// TwinCAT 3 PLC project RobotArmPLC
// ProgramVersion: 3.1.0.8
// libraries:
//   Tc2_MC2, * (Beckhoff Automation GmbH)
//   Tc2_SerialCom, * (Beckhoff Automation GmbH)
//   Tc2_Standard, * (Beckhoff Automation GmbH)
//   Tc2_System, * (Beckhoff Automation GmbH)
//   Tc3_Interfaces, * (Beckhoff Automation GmbH)
//   Tc3_Module, * (Beckhoff Automation GmbH)
// project tree:
//   GVLs/ GVL.TcGVL
//   / PlcTask.TcTTO
//   POUs/ MAIN.TcPOU, SerialRecieve.TcPOU, ShoudlerInit.TcPOU, ShoulderLevelShift.TcPOU, ShoulderRotate.TcPOU
// real-time tasks:
//   TASK PlcTask: cycle T#10ms, priority 20, ADS port 350
//   TASK CPP: cycle T#10ms, priority 1, ADS port 351
// motion (NC):
//   TASK NC-Task 1 SAF: cycle T#10ms, priority 4, ADS port 501
//   TASK NC-Task 1 SVB: cycle T#10ms, priority 8, ADS port 511
//   AXIS AxisShoulderLevelShift (id 1)
//     Velo: SlowManual=0.5, FastManual=2, Maximum=8
//     OtherSettings: AllowMotionCmdToSlave=true
//     encoder EncType=19
//       EncPara: MaxCount=#xffffffff
//     drive DrvType=16
//       DrvPara: MaxCount=#xffffffff
//         Analog: VeloReferenz=7
//         TimeComp: TaskDelayCycles=1
//     controller CtrType=1
//       CtrPara: PriorControlFactor=1
//         Observer: BandWidth=20
//   AXIS AxisShoulderRotate (id 2)
//     Velo: SlowManual=0.5, FastManual=2, Maximum=8
//     OtherSettings: AllowMotionCmdToSlave=true
//     encoder EncType=19
//       EncPara: MaxCount=#xffffffff
//     drive DrvType=16
//       DrvPara: MaxCount=#xffffffff
//         Analog: VeloReferenz=7
//         TimeComp: TaskDelayCycles=1
//     controller CtrType=1
//       CtrPara: PriorControlFactor=1
//         Observer: BandWidth=20
// I/O:
//   DEVICE Device 1 (EtherCAT), AmsNetId 5.36.3.8.2.1
//     Term 1 (EK1200) [EK1200-5000 EtherCAT Power supply (2A E-Bus)]
//       Term 2 (EL2502) [EL2502 2Ch. PWM output, 24V]
//       Term 3 (EL6001) [EL6001 Interface (RS232)]
//       Term 4 (EL4102) [EL4102 2Ch. Ana. Output  0-10V, 16bit]
//       Term 5 (EL2502) [EL2502 2K. PWM Ausgang, 24V]
//       Term 6 (EL2502) [EL2502 2Ch. PWM Output, 24V]
//       Term 7 (EL2502) [EL2502 2Ch. PWM Output, 24V]
//       Term 8 (EL3008) [EL3008 8Ch. Ana. Input +/-10V]
//       Term 9 (EL2502) [EL2502 2Ch. PWM output, 24V]
//       Term 10 (EL2502) [EL2502 2K. PWM Ausgang, 24V]
//       Term 11 (EL2502) [EL2502 2K. PWM Ausgang, 24V]
//       Term 12 (EL2502) [EL2502 2Ch. PWM output, 24V]
//       Term 13 (EL3692) [EL3692 2Ch. resistance measurement terminal]
//       Term 14 (EL9011) [EL9011 End Terminal]
//   DEVICE Device 4 (EtherCAT), AmsNetId 5.36.3.8.5.1
//     Drive 1 (Elmo Drive) [Gold EtherCAT GCON Drive Rev:0x000103F6]
//     Drive 2 (Elmo Drive) [Gold EtherCAT GCON Drive Rev:0x000103F6]
// variable links:
//   Device 1 (EtherCAT) <-> RobotArmCPP/RobotArmCPP_Obj1 (CRobotArmMain)
//     Term 1 (EK1200)/Term 10 (EL2502)/PWM Outputs Channel 1/PWM output <-> Outputs/wrist_three
//     Term 1 (EK1200)/Term 10 (EL2502)/PWM Outputs Channel 2/PWM output <-> Outputs/wrist_four
//     Term 1 (EK1200)/Term 11 (EL2502)/PWM Outputs Channel 1/PWM output <-> Outputs/wrist_five
//     Term 1 (EK1200)/Term 11 (EL2502)/PWM Outputs Channel 2/PWM output <-> Outputs/wrist_six
//     Term 1 (EK1200)/Term 12 (EL2502)/PWM Outputs Channel 1/PWM output <-> Outputs/wrist_seven
//     Term 1 (EK1200)/Term 12 (EL2502)/PWM Outputs Channel 2/PWM output <-> Outputs/wrist_eight
//     Term 1 (EK1200)/Term 13 (EL3692)/SAI Inputs Real Channel 1/Value <-> Inputs/wrist_resistor
//     Term 1 (EK1200)/Term 4 (EL4102)/Channel 1/Output <-> Outputs/ElbowOutM1
//     Term 1 (EK1200)/Term 4 (EL4102)/Channel 2/Output <-> Outputs/ElbowOutM2
//     Term 1 (EK1200)/Term 5 (EL2502)/PWM Outputs Channel 1/PWM output <-> Outputs/hand_one
//     Term 1 (EK1200)/Term 5 (EL2502)/PWM Outputs Channel 2/PWM output <-> Outputs/hand_two
//     Term 1 (EK1200)/Term 6 (EL2502)/PWM Outputs Channel 1/PWM output <-> Outputs/hand_three
//     Term 1 (EK1200)/Term 6 (EL2502)/PWM Outputs Channel 2/PWM output <-> Outputs/hand_four
//     Term 1 (EK1200)/Term 7 (EL2502)/PWM Outputs Channel 1/PWM output <-> Outputs/hand_fan
//     Term 1 (EK1200)/Term 8 (EL3008)/AI Standard Channel 1/Value <-> Inputs/hand_one_temp
//     Term 1 (EK1200)/Term 8 (EL3008)/AI Standard Channel 2/Value <-> Inputs/hand_two_temp
//     Term 1 (EK1200)/Term 8 (EL3008)/AI Standard Channel 3/Value <-> Inputs/hand_three_temp
//     Term 1 (EK1200)/Term 8 (EL3008)/AI Standard Channel 4/Value <-> Inputs/hand_four_temp
//     Term 1 (EK1200)/Term 9 (EL2502)/PWM Outputs Channel 1/PWM output <-> Outputs/wrist_one
//     Term 1 (EK1200)/Term 9 (EL2502)/PWM Outputs Channel 2/PWM output <-> Outputs/wrist_two
//   NC-Task 1 SAF/Axes/AxisShoulderLevelShift <-> Device 4 (EtherCAT)/Drive 1 (Elmo Drive)
//     Drive/Inputs/In/nDcOutputTime <-> InfoData/DcOutputShift
//     Drive/Inputs/In/nState1 <-> Inputs/Status word
//     Drive/Inputs/In/nState2 <-> Inputs/Status word @bit 8
//     Drive/Inputs/In/nState4 @bit 1 <-> WcState/InputToggle
//     Drive/Inputs/In/nState4 <-> WcState/WcState
//     Drive/Outputs/Out/nCtrl1 <-> Outputs/Control word
//     Drive/Outputs/Out/nCtrl2 <-> Outputs/Control word @bit 8
//     Drive/Outputs/Out/nDataOut1 <-> Outputs/Target Position
//     Enc/Inputs/In/nDataIn1 <-> Inputs/Position actual value
//     Enc/Inputs/In/nDcInputTime <-> InfoData/DcInputShift
//     Enc/Inputs/In/nState4 @bit 1 <-> WcState/InputToggle
//     Enc/Inputs/In/nState4 <-> WcState/WcState
//   NC-Task 1 SAF/Axes/AxisShoulderRotate <-> Device 4 (EtherCAT)/Drive 2 (Elmo Drive)
//     Drive/Inputs/In/nDcOutputTime <-> InfoData/DcOutputShift
//     Drive/Inputs/In/nState1 <-> Inputs/Status word
//     Drive/Inputs/In/nState2 <-> Inputs/Status word @bit 8
//     Drive/Inputs/In/nState4 @bit 1 <-> WcState/InputToggle
//     Drive/Inputs/In/nState4 <-> WcState/WcState
//     Drive/Outputs/Out/nCtrl1 <-> Outputs/Control word
//     Drive/Outputs/Out/nCtrl2 <-> Outputs/Control word @bit 8
//     Drive/Outputs/Out/nDataOut1 <-> Outputs/Target Position
//     Enc/Inputs/In/nDataIn1 <-> Inputs/Position actual value
//     Enc/Inputs/In/nDcInputTime <-> InfoData/DcInputShift
//     Enc/Inputs/In/nState4 @bit 1 <-> WcState/InputToggle
//     Enc/Inputs/In/nState4 <-> WcState/WcState
//   RobotArmPLC/RobotArmPLC Instance <-> Device 1 (EtherCAT)/Term 1 (EK1200)/Term 3 (EL6001)
//     PlcTask Inputs/SerialRecieve.EL6_22Bin_PC1/D <-> COM Inputs/Data In 0
//     PlcTask Inputs/SerialRecieve.EL6_22Bin_PC1/D @bit {8..168 step 8} <-> COM Inputs/Data In {1..21}  (21 links)
//     PlcTask Inputs/SerialRecieve.EL6_22Bin_PC1/Status <-> COM Inputs/Status
//     PlcTask Outputs/SerialRecieve.EL6_22Bout_PC1/Ctrl <-> COM Outputs/Ctrl
//     PlcTask Outputs/SerialRecieve.EL6_22Bout_PC1/D <-> COM Outputs/Data Out 0
//     PlcTask Outputs/SerialRecieve.EL6_22Bout_PC1/D @bit {8..168 step 8} <-> COM Outputs/Data Out {1..21}  (21 links)
//   RobotArmPLC/RobotArmPLC Instance <-> NC-Task 1 SAF/Axes/AxisShoulderLevelShift
//     PlcTask Inputs/GVL.AxisLevelShift.NcToPlc <-> Outputs/ToPlc
//     PlcTask Outputs/GVL.AxisLevelShift.PlcToNc <-> Inputs/FromPlc
//   RobotArmPLC/RobotArmPLC Instance <-> NC-Task 1 SAF/Axes/AxisShoulderRotate
//     PlcTask Inputs/GVL.AxisRotate.NcToPlc <-> Outputs/ToPlc
//     PlcTask Outputs/GVL.AxisRotate.PlcToNc <-> Inputs/FromPlc
//   RobotArmPLC/RobotArmPLC Instance <-> RobotArmCPP/RobotArmCPP_Obj1 (CRobotArmMain)
//     PlcTask Inputs/GVL.CppErrorCode <-> CppToPlc/ErrorCode
//     PlcTask Inputs/GVL.ShoulderInitStart <-> CppToPlc/ShoulderInitStart
//     PlcTask Inputs/MAIN.ElbowAngle <-> CppToPlc/ElbowAngle
//     PlcTask Inputs/MAIN.ElbowTarAngle <-> CppToPlc/ElbowTarAngle
//     PlcTask Inputs/MAIN.hand_four_pwm <-> CppToPlc/hand_four_pwm
//     PlcTask Inputs/MAIN.hand_four_temp <-> CppToPlc/hand_four_temp
//     PlcTask Inputs/MAIN.hand_one_temp <-> CppToPlc/hand_one_temp
//     PlcTask Inputs/MAIN.hand_onepwm <-> CppToPlc/hand_one_pwm
//     PlcTask Inputs/MAIN.hand_three_pwm <-> CppToPlc/hand_three_pwm
//     PlcTask Inputs/MAIN.hand_three_temp <-> CppToPlc/hand_three_temp
//     PlcTask Inputs/MAIN.hand_two_pwm <-> CppToPlc/hand_two_pwm
//     PlcTask Inputs/MAIN.hand_two_temp <-> CppToPlc/hand_two_temp
//     PlcTask Inputs/MAIN.wrist_angle <-> CppToPlc/wrist_angle
//     PlcTask Inputs/MAIN.wrist_error <-> CppToPlc/wrist_error
//     PlcTask Inputs/MAIN.wrist_pwm_out <-> CppToPlc/wrist_pwm
//     PlcTask Inputs/MAIN.wrist_tarAngle <-> CppToPlc/wrist_tarAngle
//     PlcTask Inputs/ShoulderLevelShift.TarPosLevelShift <-> CppToPlc/TarPosLevelShift
//     PlcTask Inputs/ShoulderRotate.TarPosRotate <-> CppToPlc/TarPosRotate
//     PlcTask Outputs/GVL.ChooseAction <-> PlcToCpp/ChooseAction
//     PlcTask Outputs/GVL.ExtEnabledLevelShift <-> PlcToCpp/LevelShiftExtEnabled
//     PlcTask Outputs/GVL.ExtEnabledRotate <-> PlcToCpp/RotateExtEnabled
//     PlcTask Outputs/GVL.IsRepeat <-> PlcToCpp/IsRepeat
//     PlcTask Outputs/GVL.PosLevelShift <-> PlcToCpp/PosLevelShift
//     PlcTask Outputs/GVL.PosRotate <-> PlcToCpp/PosRotate
//     PlcTask Outputs/GVL.SetTarAngle <-> PlcToCpp/SetTarAngle
//     PlcTask Outputs/GVL.SetTarSpeed <-> PlcToCpp/SetTarSpeed
//     PlcTask Outputs/GVL.ShoulderInitFinish <-> PlcToCpp/ShoulderInitFinish
//     PlcTask Outputs/GVL.StopElbow <-> PlcToCpp/StopElbow
//     PlcTask Outputs/GVL.StopHand <-> PlcToCpp/StopHand
//     PlcTask Outputs/GVL.StopWrist <-> PlcToCpp/StopWrist
//     PlcTask Outputs/GVL.Timer <-> PlcToCpp/Timer
//     PlcTask Outputs/MAIN.PlcStarted <-> PlcToCpp/PlcStarted
//     PlcTask Outputs/SerialRecieve.JIAODU <-> PlcToCpp/ElbowAngle

CONFIGURATION RobotArmPLC
    RESOURCE PLC ON TwinCAT3
        TASK PlcTask(INTERVAL := T#10ms, PRIORITY := 20);
        PROGRAM MAIN WITH PlcTask : MAIN;
        PROGRAM SerialRecieve WITH PlcTask : SerialRecieve;
        PROGRAM ShoudlerInit WITH PlcTask : ShoudlerInit;
        PROGRAM ShoulderLevelShift WITH PlcTask : ShoulderLevelShift;
        PROGRAM ShoulderRotate WITH PlcTask : ShoulderRotate;
    END_RESOURCE
END_CONFIGURATION

// ---- GVLs/GVL.TcGVL
VAR_GLOBAL
	//肩关节水平移动自由度变量
	AxisLevelShift: AXIS_REF;											//运动轴
	MC_PowerLevelShift: MC_Power;										//电源模块
	MC_MoveAbsoluteLevelShift: MC_MoveAbsolute;							//绝对运动模块
	PosLevelShift AT%Q* : LREAL;										//平移运动位置.输出给C++
	
	//肩关节旋转移动自由度变量
	AxisRotate: AXIS_REF;												//运动轴
	MC_PowerRotate: MC_Power;											//电源模块
	MC_MoveAbsoluteRotate: MC_MoveAbsolute;								//绝对运动模块
	MC_ExtSetPointGenDisableRotate: MC_ExtSetPointGenDisable;			//外部给定运动禁止
	MC_ExtSetPointGenEnableRotate: MC_ExtSetPointGenEnable;				//外部给定运动使能
	PosRotate AT%Q* : LREAL;											//旋转移动位置.输出给C++
	
	//肩关节初始化完成标志量
	ShoulderInitStart AT%I* : BOOL := FALSE;							//肩关节初始化启动
	ShoulderInitFinish AT%Q*: BOOL := FALSE;
	ExtEnabledLevelShift AT%Q* : BOOL := FALSE;							//平移外部给定模块已使能
	ExtEnabledRotate AT%Q* : BOOL := FALSE;								//旋转外部给定模块已使能
	
	//PLC时间
	Timer AT%Q*: LREAL := 0;											//时间 
	
	//错误记录
	CppErrorCode AT%I*: INT := 0;										//C++错误代码，在PLC显示，容易看到。
	ErrorCode: INT := 0;												//PLC错误代码，TODO:研究可持续写入的变量，类似字符串。
	ErrorTime: LREAL := 0;												//错误发生的时间，共4位
																		//第一位无意义，第二位表示关节（0-4：肩平移、肩旋转、肘、腕、手）
																		//第三位表示关节自由度（例如肩关节0表示平移自由度，1表示旋转自由度）
																		//第四位表示错误信息
																		//1000：平移初始化电源使能错误
																		//1001：平移位置超过限制
																		//1002：平移速度超过限制
																		//1100：旋转初始化电源使能错误
																		//1101：旋转位置超过限制
																		//1102：旋转速度超过限制
	ErrorTarPosLevelShift : LREAL := 0;									//错误发生时平移期望位置
	ErrorTarPosRotate : LREAL := 0;										//错误发生时旋转期望位置
	
	StopElbow AT%Q* : BOOL := FALSE;									//气动放气标志量，手动在plc里设置
	StopWrist AT%Q* : BOOL := FALSE;
	StopHand AT%Q* : BOOL := FALSE;
	
	ChooseAction AT%Q* : INT := -1;
	IsRepeat AT%Q* : BOOL := FALSE;
	SetTarAngle AT%Q* : LREAL := 30;									//角度定位
	SetTarSpeed AT%Q* : LREAL := 2;										//速度设置，到达100度
END_VAR

// ---- POUs/MAIN.TcPOU
PROGRAM MAIN
VAR
	ElbowTarAngle AT%I* : LREAL;
	ElbowAngle AT%I* : LREAL;
	ElbowAngleError : LREAL;
	PlcStarted AT%Q* : BOOL := FALSE;
	
	wrist_pwm_out AT%I*: LREAL;
	wrist_angle AT%I*: LREAL;
	wrist_tarAngle AT%I*: LREAL;
	wrist_error AT%I*: LREAL;
	flag_plc AT%Q*: BOOL;
///////////////腕关节变量监测/////
	
	hand_one_temp AT%I*: INT;
	hand_two_temp AT%I*: INT;
	hand_three_temp AT%I*: INT;
	hand_four_temp AT%I*: INT;
	hand_onepwm AT%I*: INT;
	hand_two_pwm AT%I*: INT;
	hand_three_pwm AT%I*: INT;
	hand_four_pwm AT%I*: INT;
/////////////手部变量监测/////////
END_VAR

//PlcStarted := TRUE;

(*IF InitFinish AND ExtEnabledLevelShift AND ExtEnabledRotate THEN
	Timer := Timer + 0.01;
END_IF*)
Timer := Timer + 0.01;

ElbowAngleError := ElbowTarAngle - ElbowAngle;
wrist_error := wrist_tarAngle - wrist_angle;

END_PROGRAM

// ---- POUs/SerialRecieve.TcPOU
PROGRAM SerialRecieve
VAR
	//读取编码器角度
	EL6_22Bin_PC1	AT %I* 	: KL6inData22b;
	EL6_22Bout_PC1	AT %Q*	: KL6outData22b;
	RxBuffer1: COMBuffer;
	TxBuffer1: COMBuffer;
	JIAODU	AT %Q* : LREAL;(*单位 度*)
	JIAOSUDU: LREAL;(*单位 度*)
	JIAOJIASUDU: LREAL;(*单位 度*)
	SerialLineControlElbow:SerialLineControl;
	
	i:INT;
    AA:BYTE;
	BB:BYTE;
	RxBufferStep:INT:=0;
    AA_P:BYTE;
	BB_P:BYTE;
	JIAODU_INT:INT;
	J1: LREAL:=0;
	J2: LREAL:=0;
	J3: LREAL:=0;
	W1: LREAL:=0;
	W2: LREAL:=0;
	t_tip: LREAL:=0.01;
END_VAR

//读取编码器的数值
SerialLineControlElbow(
	Mode:= SERIALLINEMODE_KL6_22B_STANDARD, 
	pComIn:= ADR(EL6_22Bin_PC1), 
	pComOut:= ADR(EL6_22Bout_PC1), 
	SizeComIn:= UINT_TO_INT(SIZEOF(EL6_22Bin_PC1)), 
	TxBuffer:= TxBuffer1, 
	RxBuffer:= RxBuffer1);

IF RxBuffer1.Count<> 0 THEN
	FOR i:=1 TO UINT_TO_INT(RxBuffer1.Count) DO
		IF RxBufferStep=3 THEN
			BB:=RxBuffer1.Buffer[RxBuffer1.RdIdx];
			AA:=AA_P;
			RxBufferStep:=0;
		END_IF
		IF RxBufferStep=2 THEN
			AA_P:=RxBuffer1.Buffer[RxBuffer1.RdIdx];
			RxBufferStep:=3;
		END_IF
		IF RxBufferStep=1 THEN
			IF RxBuffer1.Buffer[RxBuffer1.RdIdx]=90 THEN
				RxBufferStep:=2;
			ELSE
				RxBufferStep:=0;
			END_IF
		END_IF
		IF RxBuffer1.Buffer[RxBuffer1.RdIdx]=165 THEN
			RxBufferStep:=1;
		END_IF

		RxBuffer1.RdIdx:=RxBuffer1.RdIdx+1;
		IF RxBuffer1.RdIdx>300 THEN
			RxBuffer1.RdIdx:=0;
		END_IF
	END_FOR
RxBuffer1.Count:=0;
END_IF

JIAODU_INT:=UINT_TO_INT(AA*256+BB);
JIAODU:=INT_TO_REAL(JIAODU_INT)*360.0/4096.0;
J3:=J2;
J2:=J1;
J1:=JIAODU;
JIAOSUDU:=(J1-J2)/t_tip;
W2:=W1;
W1:=JIAOSUDU;
JIAOJIASUDU:=(W1-W2)/t_tip;

END_PROGRAM

// ---- POUs/ShoudlerInit.TcPOU
PROGRAM ShoudlerInit
VAR
	InitPosLevelShift: LREAL := 0;			//平移自由度.初始化位置
	InitStatusLevelShift: INT := 0;			//平移自由度.初始化状态变量	
	InitFinishLevelShift: BOOL := FALSE;	//平移自由度.初始化完成标志量
	
	InitPosRotate: LREAL := 0;				//旋转自由度.初始化位置
	InitStatusRotate: INT := 0;				//旋转自由度.初始化状态变量	
	InitFinishRotate: BOOL := FALSE;		//旋转自由度.初始化完成标志量
END_VAR

//肩关节初始化

//平移自由度
MC_PowerLevelShift(
	Axis:= AxisLevelShift,
	Enable_Positive:= TRUE,
	Enable_Negative:= TRUE, );
	
MC_MoveAbsoluteLevelShift(
	Axis:= AxisLevelShift, );

CASE InitStatusLevelShift OF
	0://等待初始化命令
		IF ShoulderInitStart THEN
			InitStatusLevelShift := 1;
		END_IF
	1://init 初始化
		MC_PowerLevelShift.Enable := FALSE;
		MC_MoveAbsoluteLevelShift.Execute := FALSE;
		InitStatusLevelShift := 2;
	2://power 使能
		MC_PowerLevelShift.Enable := TRUE;
		IF MC_PowerLevelShift.Status THEN
			InitStatusLevelShift := 3;
		END_IF
		IF AxisLevelShift.Status.Error THEN
			ErrorTime := Timer;
			InitStatusLevelShift := 5;
		END_IF
	3://move 移动到初始位置
		MC_MoveAbsoluteLevelShift.Position := InitPosLevelShift;
		MC_MoveAbsoluteLevelShift.Velocity := 1;
		MC_MoveAbsoluteLevelShift.Execute := TRUE;
		IF MC_MoveAbsoluteLevelShift.Done THEN
			MC_MoveAbsoluteLevelShift.Execute := FALSE;
			InitStatusLevelShift := 4;
		END_IF
	4://finishInit 初始化完成
		InitFinishLevelShift := TRUE;
	5://error
		ErrorCode := 1000;
END_CASE


//旋转自由度
MC_PowerRotate(
	Axis:= AxisRotate,
	Enable_Positive:= TRUE,
	Enable_Negative:= TRUE, );
	
MC_MoveAbsoluteRotate(
	Axis:= AxisRotate, );

CASE InitStatusRotate OF
	0://等待初始化命令
		IF ShoulderInitStart THEN
			InitStatusRotate := 1;
		END_IF
	1://init 初始化
		MC_PowerRotate.Enable := FALSE;
		MC_MoveAbsoluteRotate.Execute := FALSE;
		InitStatusRotate := 2;
	2://power 使能
		MC_PowerRotate.Enable := TRUE;
		IF MC_PowerRotate.Status THEN
			InitStatusRotate := 3;
		END_IF
		IF AxisLevelShift.Status.Error THEN
			ErrorTime := Timer;
			InitStatusRotate := 5;
		END_IF
	3://move 移动到初始位置
		MC_MoveAbsoluteRotate.Position := InitPosLevelShift;
		MC_MoveAbsoluteRotate.Velocity := 1;
		MC_MoveAbsoluteRotate.Execute := TRUE;
		IF MC_MoveAbsoluteRotate.Done THEN
			MC_MoveAbsoluteRotate.Execute := FALSE;
			InitStatusRotate := 4;
		END_IF
	4://finishInit 初始化完成
		InitFinishRotate := TRUE;
	5://error
		ErrorCode := 1100;
END_CASE
		
IF InitFinishLevelShift AND InitFinishRotate THEN
	ShoulderInitFinish := TRUE;
END_IF

END_PROGRAM

// ---- POUs/ShoulderLevelShift.TcPOU
PROGRAM ShoulderLevelShift
VAR
	MC_ExtSetPointGenDisableLevelShift: MC_ExtSetPointGenDisable;		//外部给定运动禁止
	MC_ExtSetPointGenEnableLevelShift: MC_ExtSetPointGenEnable;			//外部给定运动使能
	
	//TODO: C++将目标角度转换为目标位置
	TarPosLevelShift AT%I* : LREAL := 0;								//平移目标位置，C++给定
	ErrPosLevelShift: LREAL := 0;										//目标位置和实际位置误差
	
	StatusLevelShift: INT := 0;											//状态变量
	
	test : LREAL := 0;
END_VAR

//肩关节水平移动自由度

//电机外部给定运动模块参数设置
MC_ExtSetPointGenDisableLevelShift(
	Axis:= AxisLevelShift, );
	
MC_ExtSetPointGenEnableLevelShift(
	Axis:= AxisLevelShift, );
	
PosLevelShift := AxisLevelShift.NcToPlc.ActPos;

CASE StatusLevelShift OF
	0:	//判断是否完成初始化
		IF ShoulderInitFinish THEN
			StatusLevelShift := 1;
		END_IF
	1:	//外部给定模块使能给低电平
		MC_ExtSetPointGenEnableLevelShift.Execute := FALSE;
		MC_ExtSetPointGenDisableLevelShift.Execute := FALSE;
		StatusLevelShift := 2;
	2:
		MC_ExtSetPointGenEnableLevelShift.Execute := TRUE;
		IF MC_ExtSetPointGenEnableLevelShift.Enabled THEN
			StatusLevelShift := 3;
			ExtEnabledLevelShift := TRUE;
		END_IF
	3:	//判断目标移动是否有问题
		//Timer := Timer + 0.01;
		IF TarPosLevelShift > 18 OR TarPosLevelShift < -15 THEN
			ErrorCode := 1001;
			ErrorTime := Timer;
			StatusLevelShift := 4;						//跳转到错误处理状态
		END_IF
		ErrPosLevelShift := TarPosLevelShift - AxisLevelShift.NcToPlc.ActPos;//误差:目标角度减去实际角度
//		IF ABS(ErrPosLevelShift) < 1E-8 THEN			//移动距离过小认为不移动
			//不移动
//		ELSIF ABS(ErrPosLevelShift) > 0.15 THEN
		IF ABS(ErrPosLevelShift) > 0.15 THEN
			//安全保护。单次移动距离过大，即移动速度过快，停止运动。
			//|maxV| = 15 mm/s; |maxv| = 0.15 mm / 0.01s;
			ErrorCode := 1002;
			ErrorTime := Timer;
			ErrorTarPosLevelShift := TarPosLevelShift;
			StatusLevelShift := 4;						//跳转到错误处理状态
		ELSE											//按照给定移动
			IF MC_ExtSetPointGenEnableLevelShift.Enabled THEN
				MC_ExtSetPointGenFeed(
					//Position:= Timer,		//给定位置
					Position:= TarPosLevelShift,		//给定位置
					Velocity:= 0, 						//速度和加速度可设为0，让plc自己计算
					Acceleration:= 0, 
					Direction:= 1, 
					Axis:= AxisLevelShift);
			END_IF
		END_IF
	4:	//Error处理
		MC_ExtSetPointGenEnableLevelShift.Execute := FALSE;	//关闭外部位置给定
		MC_ExtSetPointGenDisableLevelShift.Execute := TRUE;
END_CASE

END_PROGRAM

// ---- POUs/ShoulderRotate.TcPOU
PROGRAM ShoulderRotate
VAR
	MC_ExtSetPointGenDisableRotate: MC_ExtSetPointGenDisable;
	MC_ExtSetPointGenEnable: MC_ExtSetPointGenEnable;
	
	TarPosRotate AT%I* : LREAL := 0;
	ErrPosRotate: LREAL := 0;										//目标位置和实际位置误差
	
	StatusRotate: INT := 0;											//状态变量

END_VAR

//肩关节旋转移动自由度

//电机外部给定运动模块参数设置
MC_ExtSetPointGenDisableRotate(
	Axis:= AxisRotate, );
	
MC_ExtSetPointGenEnableRotate(
	Axis:= AxisRotate, );
	
PosRotate := AxisRotate.NcToPlc.ActPos;

CASE StatusRotate OF
	0:	//判断是否完成初始化
		IF ShoulderInitFinish THEN
			StatusRotate := 1;
		END_IF
	1:	//外部给定模块使能给低电平
		MC_ExtSetPointGenEnableRotate.Execute := FALSE;
		MC_ExtSetPointGenDisableRotate.Execute := FALSE;
		StatusRotate := 2;
	2:
		MC_ExtSetPointGenEnableRotate.Execute := TRUE;
		IF MC_ExtSetPointGenEnableRotate.Enabled THEN
			StatusRotate := 3;
			ExtEnabledRotate := TRUE;
		END_IF
	3:	//判断目标移动是否有问题
		//Timer := Timer + 0.01;
		IF TarPosRotate > 15 OR TarPosRotate < -15 THEN
			ErrorCode := 1011;
			ErrorTime := Timer;
			StatusRotate := 4;						//跳转到错误处理状态
		END_IF
		ErrPosRotate := TarPosRotate - AxisRotate.NcToPlc.ActPos;//误差:目标角度减去实际角度
//		IF ABS(ErrPosRotate) < 1E-8 THEN			//移动距离过小认为不移动
			//不移动
//		ELSIF ABS(ErrPosRotate) > 0.15 THEN
		IF ABS(ErrPosRotate) > 0.15 THEN
			//安全保护。单次移动距离过大，即移动速度过快，停止运动。
			//|maxV| = 15 mm/s; |maxv| = 0.15 mm / 0.01s;
			ErrorCode := 1012;
			ErrorTime := Timer;
			ErrorTarPosRotate := TarPosRotate;
			StatusRotate := 4;						//跳转到错误处理状态
		ELSE											//按照给定移动
			IF MC_ExtSetPointGenEnableRotate.Enabled THEN
				MC_ExtSetPointGenFeed(
					//Position:= Timer,		//给定位置
					Position:= TarPosRotate,		//给定位置
					Velocity:= 0, 						//速度和加速度可设为0，让plc自己计算
					Acceleration:= 0, 
					Direction:= 1, 
					Axis:= AxisRotate);
			END_IF
		END_IF
	4:	//Error处理
		MC_ExtSetPointGenEnableRotate.Execute := FALSE;	//关闭外部位置给定
		MC_ExtSetPointGenDisableRotate.Execute := TRUE;
END_CASE

END_PROGRAM
